PROGRAM Connect
VAR
	Connect_R1			:FB_Verbinden;
	Connect_R2			:FB_Verbinden;
	Connect_R3			:FB_Verbinden;
	Connect_R4			:FB_Verbinden;
	Connect_R5			:FB_Verbinden;
	Connect_R6			:FB_Verbinden;
	Connect_R7			:FB_Verbinden;
END_VAR

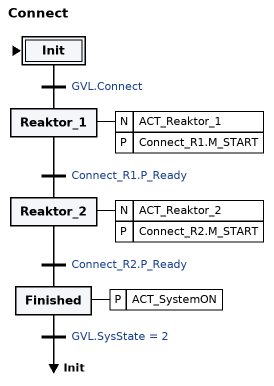
INITIAL_STEP Init:
END_STEP
TRANSITION FROM Init TO Reaktor_1
    := GVL.Connect;
END_TRANSITION
STEP Reaktor_1:
    ACT_Reaktor_1(N);
    Connect_R1.M_START(P);
END_STEP
TRANSITION FROM Reaktor_1 TO Reaktor_2
    := Connect_R1.P_Ready;
END_TRANSITION
STEP Reaktor_2:
    ACT_Reaktor_2(N);
    Connect_R2.M_START(P);
END_STEP
TRANSITION FROM Reaktor_2 TO Finished_
    := Connect_R2.P_Ready;
END_TRANSITION
STEP Finished_:  // name as stored: Finished 
    ACT_SystemON(P);
END_STEP
TRANSITION FROM Finished_ TO Init
    := GVL.SysState = 2;
END_TRANSITION

ACTION ACT_Reaktor_1:
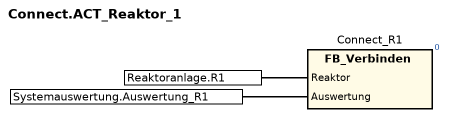
Connect_R1(Reaktor := Reaktoranlage.R1, Auswertung := Systemauswertung.Auswertung_R1); // FB_Verbinden
END_ACTION

ACTION ACT_Reaktor_2:
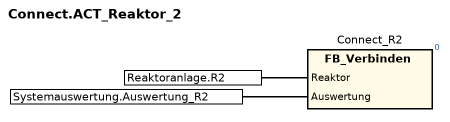
Connect_R2(Reaktor := Reaktoranlage.R2, Auswertung := Systemauswertung.Auswertung_R2); // FB_Verbinden
END_ACTION

ACTION ACT_SystemON:
GVL.SysState := 2;
END_ACTION

END_PROGRAM

(* stored: Version 1.1.0.1, ProductVersion 3.1.4024.12
   POU Connect: Id {6f9caf3c-7716-4ebf-9ccc-daf569aad75b}, SpecialFunc None
   Action ACT_Reaktor_1: Id {c780a2d0-cb1f-4bcc-8cbc-d9ba70321e8c}
   Action ACT_Reaktor_2: Id {687dd86e-7183-4468-a09d-d406dc2f1b71}
   Action ACT_SystemON: Id {15eb8c36-0b5a-47f1-9dcf-fd1ea5556748} *)
